TYPE ST_HW_OutputsTurnTable :

STRUCT
	//Turn table outputs
	Drive_Run_CW		: BOOL; // Drive run command turn table clockwise
	Drive_Run_CCW		: BOOL; // Drive run command turn table counter-clockwise
	//Drive_Low_CW_CCW	: BOOL; // Drive slow speed command turn table
	Drive_Creep_CW_CCW	: BOOL; // Drive creep speed command turn table
	Drive_Brake_CW_CCW 	: BOOL; // Drive brake release command for turn table drive unit
		
END_STRUCT
END_TYPE

(* stored: Version 1.1.0.1, ProductVersion 3.1.4024.9
   DUT ST_HW_OutputsTurnTable: Id {e0d6ccd5-e66c-44c1-ada9-d6984e388bbb} *)
